(* IEC 61131-3 sources: volt/packages/volt-lsp-iec/test-corpus/pro2193/Device/Plc Logic/Application/09 Misc/Library Manager/CAA TickUtil, 8 files *)

(* ---- VERSIONCONSTANTS.gvl ---- *)
VAR_GLOBAL
	GC_BYVERSION : BYTE := 1;
	GC_VERSION_1 : BYTE := 0;
END_VAR

(* ---- CONVERTNSECTOTICK.pou ---- *)
FUNCTION CONVERTNSECTOTICK : CAA.TICK
VAR_INPUT
	UDINSECONDS : UDINT;
END_VAR
END_FUNCTION

(* ---- CONVERTTICKTONSEC.pou ---- *)
FUNCTION CONVERTTICKTONSEC : UDINT
VAR_INPUT
	TKTICK : CAA.TICK;
END_VAR
END_FUNCTION

(* ---- CONVERTTICKTOUSEC.pou ---- *)
FUNCTION CONVERTTICKTOUSEC : UDINT
VAR_INPUT
	TKTICK : CAA.TICK;
END_VAR
END_FUNCTION

(* ---- CONVERTUSECTOTICK.pou ---- *)
FUNCTION CONVERTUSECTOTICK : CAA.TICK
VAR_INPUT
	UDIUSECONDS : UDINT;
END_VAR
END_FUNCTION

(* ---- GETELAPSEDTIMEINNSEC.pou ---- *)
FUNCTION GETELAPSEDTIMEINNSEC : UDINT
VAR_INPUT
	TKSTART : CAA.TICK;
END_VAR
END_FUNCTION

(* ---- GETELAPSEDTIMEINUSEC.pou ---- *)
FUNCTION GETELAPSEDTIMEINUSEC : UDINT
VAR_INPUT
	TKSTART : CAA.TICK;
END_VAR
END_FUNCTION

(* ---- GETSUPPLIERVERSION.pou ---- *)
FUNCTION GETSUPPLIERVERSION : WORD
VAR_INPUT
	XDUMMY : BOOL;
END_VAR
END_FUNCTION
